PROGRAM MAIN
VAR
	fbAxis					: ARRAY[1..3] OF FB_AxisPTP;
	nAnalogInput AT %I*		: INT;
	bDigitalInput AT %I*	: ARRAY[1..3] OF BOOL;
	
	eState					: (INIT, READY, RUN);
	fVelocity				: LREAL;
	bRun					: BOOL;
	i						: INT;
END_VAR

fVelocity := INT_TO_LREAL(nAnalogInput) / 32767 * 2000;

FOR i := 1 TO 3 DO
	bRun := bDigitalInput[i];
	CASE eState OF
		INIT:
			fbAxis[i].M_Invoke(FALSE);
		READY:
			fbAxis[i].M_Invoke(TRUE);
		RUN:
			fbAxis[i].fVelocity := fVelocity;
			fbAxis[i].M_MoveFw(bRun);
			fbAxis[i].M_Halt(NOT bRun);
	END_CASE
END_FOR

END_PROGRAM

(* stored: Version 1.1.0.1, ProductVersion 3.1.4024.6
   POU MAIN: Id {41904e0e-59ab-42ff-a9d4-1dc6adad7d5b}, SpecialFunc None *)
